{attribute 'qualified_only'}
VAR_GLOBAL CONSTANT

	TRACK_LENGTH 			: LREAL := 4000; // This should be set to the exact length [mm] of the track system
		
	NUM_MOVERS   			: USINT := 20;   // This should be set to the exact number of movers on the system
	
	// The following should be set to a value **equal to or greater than** the number of objectives needed
	NUM_MOVERLISTS			: USINT := 10;	// Mover Lists
	NUM_POSITIONTRIGGERS	: USINT := 10;	// Position Triggers
	NUM_STATIONS			: USINT := 10;	// Stations
	NUM_ZONES				: USINT := 10;	// Zones
	
	NUM_TRACKS				: USINT	:= 1;	// Tracks (Typically 1)

    {attribute 'TcInitSymbol'}
    pXtsProcessingUnit : OTCID:=0; // This pointer needs to be initialized in the Main Instance, under Symbol Initialization
	PART_ARRAY_SIZE			: UDINT := 100;
	AUTO_POPULATE_STATIONS  : BOOL := TRUE; // use the Station[x] array to label stations on the visualization. Turn off if manually entering stations in the configurator.
	
	// statistics weighted average
	ALPHA_EMA				: LREAL := 0.1;

END_VAR
VAR_GLOBAL
	newCallTime: LREAL;
END_VAR

(* stored: Version 1.1.0.1, ProductVersion 3.1.4024.12
   GVL GVL: Id {73e6a867-4426-4dae-a583-2a717b275c1c} *)
